// Mitsubishi GX Works2 project: NEW_PLC   PLC: FX3S

PROGRAM IN_OUT
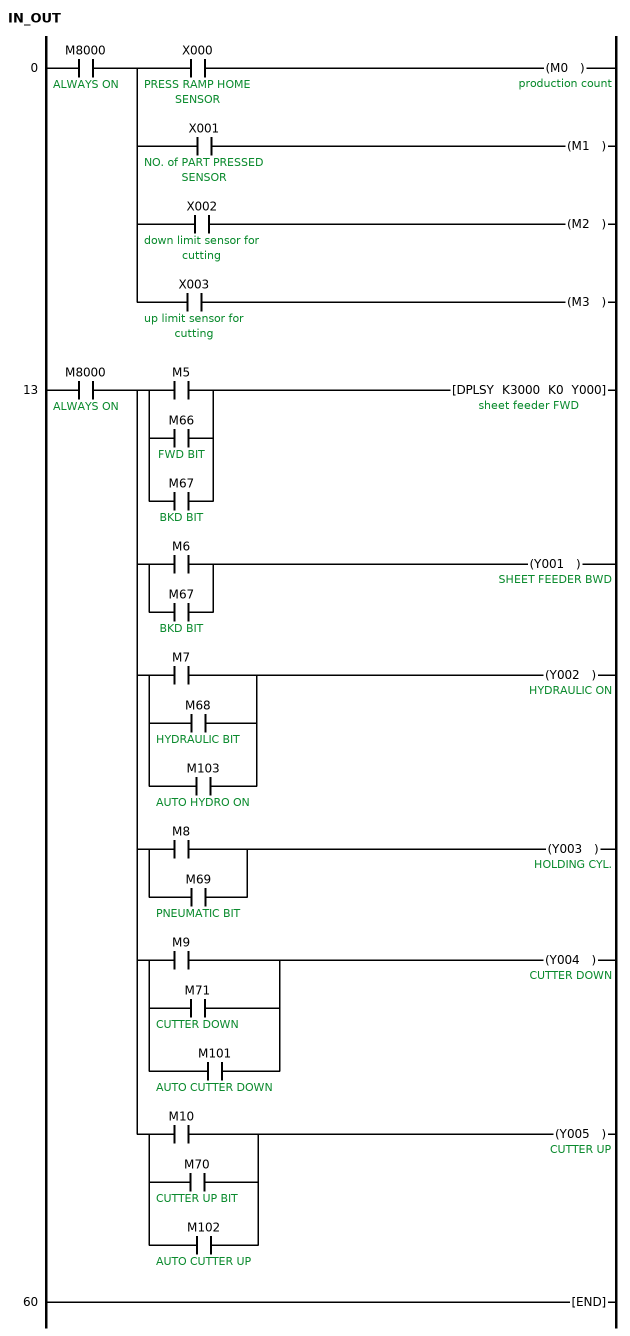
0     LD      M8000  ; ALWAYS ON
      MPS
      AND     X000  ; PRESS RAMP HOME SENSOR
      OUT     M0  ; production count
      MRD
      AND     X001  ; NO. of PART PRESSED SENSOR
      OUT     M1
      MRD
      AND     X002  ; down limit sensor for cutting
      OUT     M2
      MPP
      AND     X003  ; up limit sensor for cutting
      OUT     M3
13    LD      M8000  ; ALWAYS ON
      MPS
      LD      M5
      OR      M66  ; FWD BIT
      OR      M67  ; BKD BIT
      ANB
      DPLSY   K3000 K0 Y000  ; sheet feeder FWD
      MRD
      LD      M6
      OR      M67  ; BKD BIT
      ANB
      OUT     Y001  ; SHEET FEEDER BWD
      MRD
      LD      M7
      OR      M68  ; HYDRAULIC BIT
      OR      M103  ; AUTO HYDRO ON
      ANB
      OUT     Y002  ; HYDRAULIC ON
      MRD
      LD      M8
      OR      M69  ; PNEUMATIC BIT
      ANB
      OUT     Y003  ; HOLDING CYL.
      MRD
      LD      M9
      OR      M71  ; CUTTER DOWN
      OR      M101  ; AUTO CUTTER DOWN
      ANB
      OUT     Y004  ; CUTTER DOWN
      MPP
      LD      M10
      OR      M70  ; CUTTER UP BIT
      OR      M102  ; AUTO CUTTER UP
      ANB
      OUT     Y005  ; CUTTER UP
60    END
END_PROGRAM

PROGRAM MANUAL
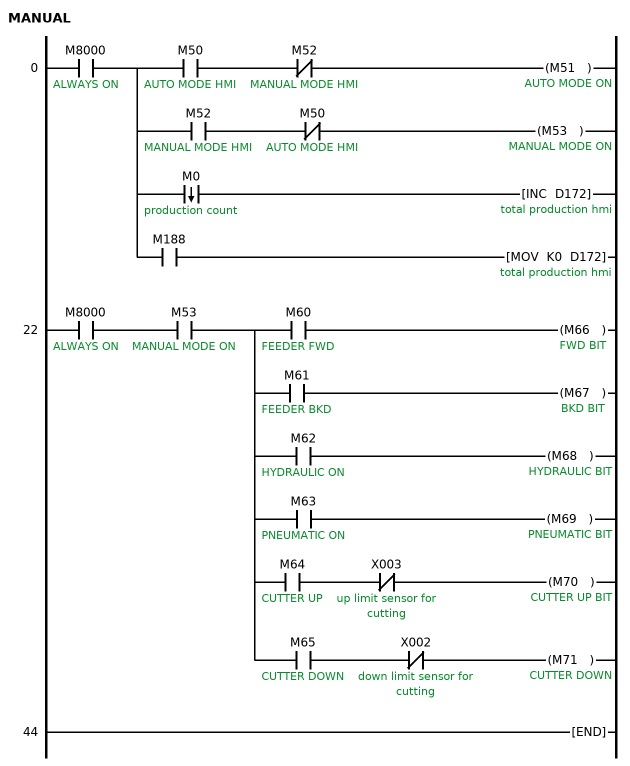
0     LD      M8000  ; ALWAYS ON
      MPS
      AND     M50  ; AUTO MODE HMI
      ANI     M52  ; MANUAL MODE HMI
      OUT     M51  ; AUTO MODE ON
      MRD
      AND     M52  ; MANUAL MODE HMI
      ANI     M50  ; AUTO MODE HMI
      OUT     M53  ; MANUAL MODE ON
      MRD
      ANDF    M0  ; production count
      INC     D172  ; total production hmi
      MPP
      AND     M188
      MOV     K0 D172
22    LD      M8000  ; ALWAYS ON
      AND     M53  ; MANUAL MODE ON
      MPS
      AND     M60  ; FEEDER FWD
      OUT     M66  ; FWD BIT
      MRD
      AND     M61  ; FEEDER BKD
      OUT     M67  ; BKD BIT
      MRD
      AND     M62  ; HYDRAULIC ON
      OUT     M68  ; HYDRAULIC BIT
      MRD
      AND     M63  ; PNEUMATIC ON
      OUT     M69  ; PNEUMATIC BIT
      MRD
      AND     M64  ; CUTTER UP
      ANI     X003  ; up limit sensor for cutting
      OUT     M70  ; CUTTER UP BIT
      MPP
      AND     M65  ; CUTTER DOWN
      ANI     X002  ; down limit sensor for cutting
      OUT     M71  ; CUTTER DOWN
44    END
END_PROGRAM

PROGRAM AUTO
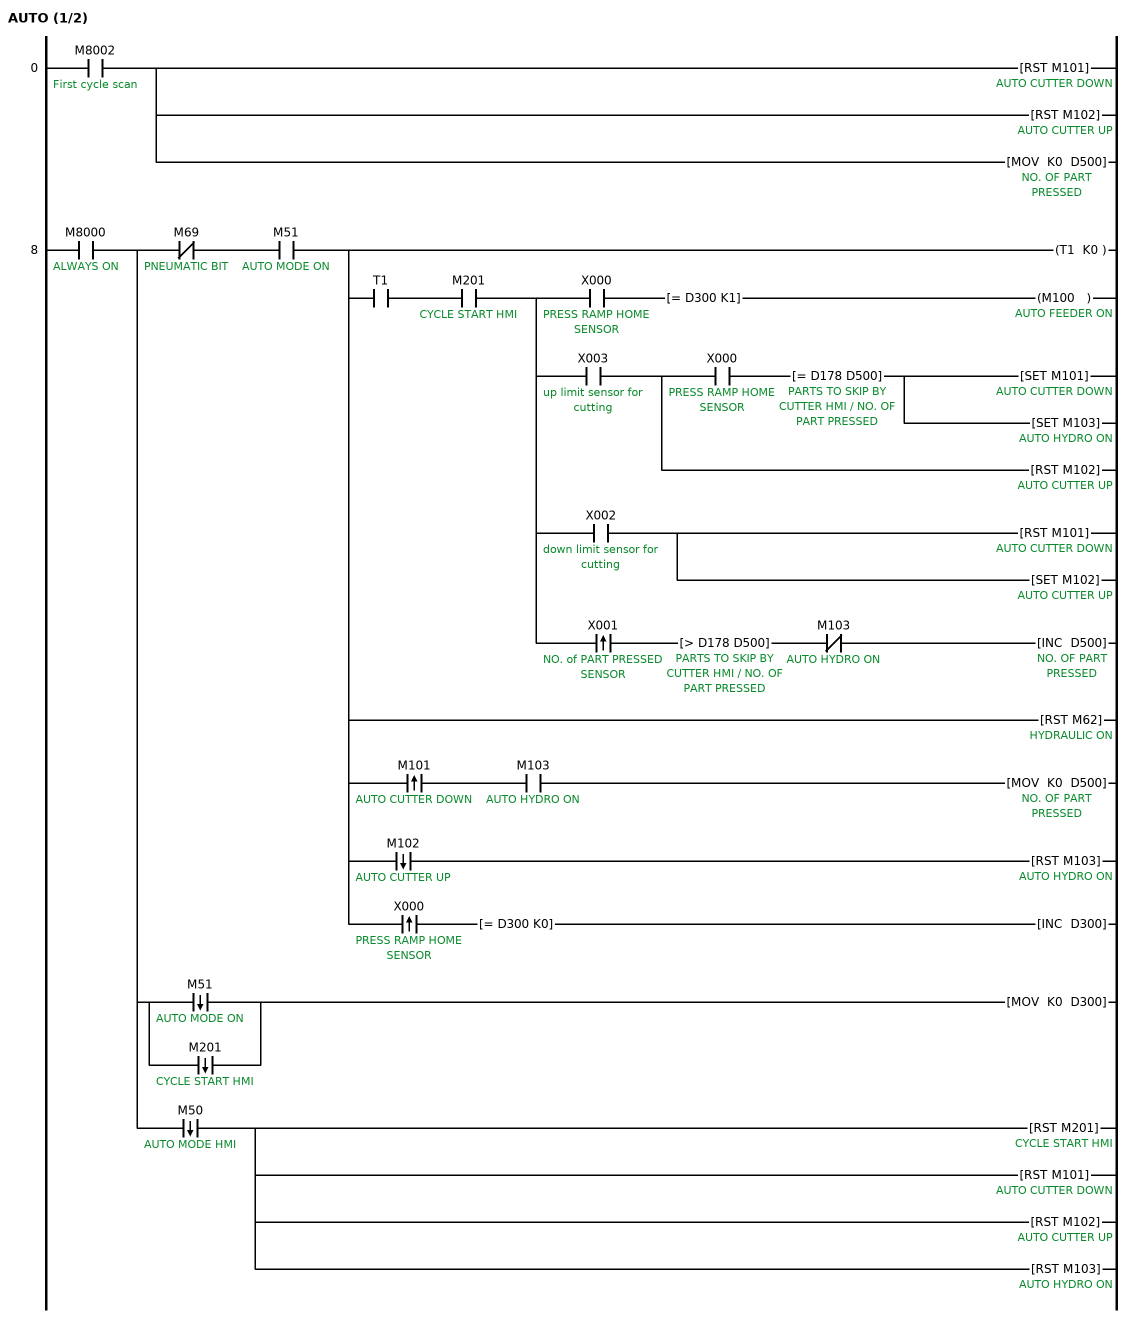
0     LD      M8002  ; First cycle scan
      RST     M101  ; AUTO CUTTER DOWN
      RST     M102  ; AUTO CUTTER UP
      MOV     K0 D500  ; NO. OF PART PRESSED
8     LD      M8000  ; ALWAYS ON
      MPS
      ANI     M69  ; PNEUMATIC BIT
      AND     M51  ; AUTO MODE ON
      OUT     T1 K0
      MPS
      AND     T1
      AND     M201  ; CYCLE START HMI
      MPS
      AND     X000  ; PRESS RAMP HOME SENSOR
      AND=    D300 K1
      OUT     M100  ; AUTO FEEDER ON
      MRD
      AND     X003  ; up limit sensor for cutting
      MPS
      AND     X000  ; PRESS RAMP HOME SENSOR
      AND=    D178 D500  ; PARTS TO SKIP BY CUTTER HMI / NO. OF PART PRESSED
      SET     M101  ; AUTO CUTTER DOWN
      SET     M103  ; AUTO HYDRO ON
      MPP
      RST     M102  ; AUTO CUTTER UP
      MRD
      AND     X002  ; down limit sensor for cutting
      RST     M101  ; AUTO CUTTER DOWN
      SET     M102  ; AUTO CUTTER UP
      MPP
      ANDP    X001  ; NO. of PART PRESSED SENSOR
      AND>    D178 D500  ; PARTS TO SKIP BY CUTTER HMI / NO. OF PART PRESSED
      ANI     M103  ; AUTO HYDRO ON
      INC     D500
      MPP
      RST     M62  ; HYDRAULIC ON
      MPS
      ANDP    M101  ; AUTO CUTTER DOWN
      AND     M103  ; AUTO HYDRO ON
      MOV     K0 D500
      MRD
      ANDF    M102  ; AUTO CUTTER UP
      RST     M103  ; AUTO HYDRO ON
      MPP
      ANDP    X000  ; PRESS RAMP HOME SENSOR
      AND=    D300 K0
      INC     D300
      MRD
      LDF     M51  ; AUTO MODE ON
      ORF     M201  ; CYCLE START HMI
      ANB
      MOV     K0 D300
      MPP
      ANDF    M50  ; AUTO MODE HMI
      RST     M201  ; CYCLE START HMI
      RST     M101  ; AUTO CUTTER DOWN
      RST     M102  ; AUTO CUTTER UP
      RST     M103  ; AUTO HYDRO ON
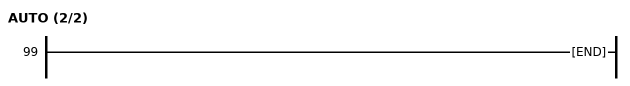
99    END
END_PROGRAM

PROGRAM servo
VAR
  flt2int : BOOL;
END_VAR
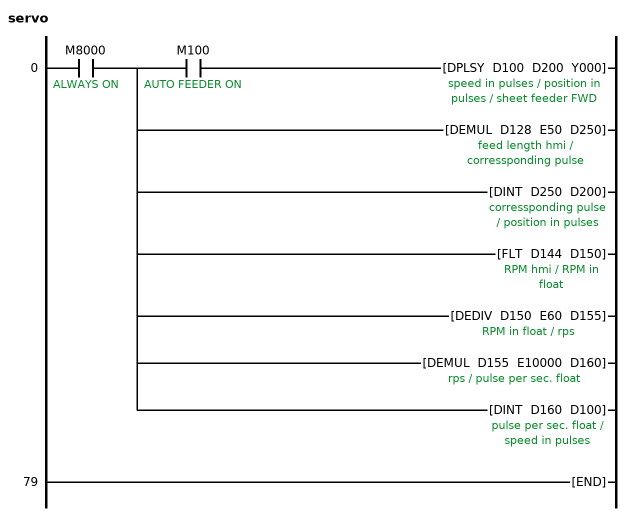
0     LD      M8000  ; ALWAYS ON
      MPS
      AND     M100  ; AUTO FEEDER ON
      DPLSY   D100 D200 Y000  ; speed in pulses / position in pulses / sheet feeder FWD
      MPP
      DEMUL   D128 E50 D250  ; feed length hmi / corressponding pulse
      DINT    D250 D200
      FLT     D144 D150  ; RPM hmi / RPM in float
      DEDIV   D150 E60 D155  ; rps
      DEMUL   D155 E10000 D160  ; pulse per sec. float
      DINT    D160 D100
79    END
END_PROGRAM

// device comments not shown above
X004  ; mould sensor(when to feed sheet)
X005  ; FOOT SWITCH TO ALLOW FEEDING
M104  ; AUTO PNEUMATIC ON
